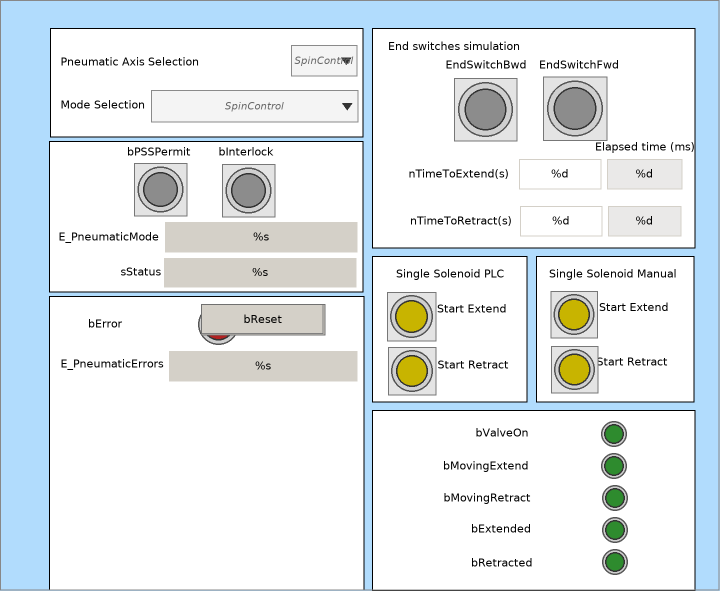
VISUALIZATION PneumaticsVisu_1  // 720x591
    Rectangle (50,28 313x109)
    Label (55,47 150x30), "Pneumatic Axis Selection"
    Rectangle (372,28 323x220)
    Label (379,30 150x33), "End switches simulation"
    Label (411,50 150x30), "EndSwitchBwd"
    SpinControl (291,45 66x31), variable: MAIN.hmiPneumaticAxisSelection
        p651134158: GVL_APP.nPNEUMATIC_AXIS_NUM
    Label (504,50 150x30), "EndSwitchFwd"
    Rectangle (49,296 315x294)
    Textfield (519,159 82x30), "%d", text variable: MAIN.afbPneumaticAxes[MAIN.hmiPneumaticAxisSelection].stPneumaticAxisStruct.stPneumaticAxisConfig.nTimeToExtend
        OnMouseClick: write MAIN.afbPneumaticAxes[MAIN.hmiPneumaticAxisSelection].stPneumaticAxisStruct.stPneumaticAxisConfig.nTimeToExtend via Default
    Label (384,159 150x30), "nTimeToExtend(s)"
    Label (386,206 150x30), "nTimeToRetract(s)"
    Label (28,90 150x30), "Mode Selection"
    Rectangle (49,141 314x151)
    Label (30,309 150x30), "bError"
    Lamp1 (126,301 185x47), variable: MAIN.afbPneumaticAxes[MAIN.hmiPneumaticAxisSelection].stPneumaticAxisStruct.stPneumaticAxisStatus.bError, style: Lamp-Lamp1-Red
    Label (37,349 150x30), "E_PneumaticErrors"
    Textfield (169,351 188x30), "%s", text variable: MAIN.afbPneumaticAxes[MAIN.hmiPneumaticAxisSelection].stPneumaticAxisStruct.ePneumaticAxisErrors, text list: 'languageSupport'
    Rectangle (372,256 155x146)
    Rectangle (536,256 158x146)
    Rectangle (372,410 323x181)
    Label (538,259 150x30), "Single Solenoid Manual"
    PushSwitchLed (549,291 50x47), variable: MAIN.afbPneumaticAxes[MAIN.hmiPneumaticAxisSelection].stPneumaticAxisStruct.stPneumaticAxisInputs.bOpenManual, behaviour: TOGGLE, style: Switch-PushSwitchLed-Yellow
    Label (592,293 84x29), "Start Extend"
    Label (557,347 150x30), "Start Retract"
    Label (375,259 150x30), "Single Solenoid PLC"
    PushSwitchLed (387,292 49x49), variable: MAIN.afbPneumaticAxes[MAIN.hmiPneumaticAxisSelection].stPneumaticAxisStruct.stPneumaticAxisControl.bExtend, behaviour: TOGGLE, style: Switch-PushSwitchLed-Yellow
    PushSwitchLed (388,347 48x48), variable: MAIN.afbPneumaticAxes[MAIN.hmiPneumaticAxisSelection].stPneumaticAxisStruct.stPneumaticAxisControl.bRetract, behaviour: TOGGLE, style: Switch-PushSwitchLed-Yellow
    Label (427,418 150x30), "bValveOn"
    Lamp1 (539,419 150x30), variable: MAIN.afbPneumaticAxes[MAIN.hmiPneumaticAxisSelection].stPneumaticAxisStruct.stPneumaticAxisOutputs.bValveOn, style: Lamp-Lamp1-Green
    Label (411,451 150x30), "bMovingExtend"
    Lamp1 (539,451 150x30), variable: MAIN.afbPneumaticAxes[MAIN.hmiPneumaticAxisSelection].stPneumaticAxisStruct.stPneumaticAxisStatus.bExtending, style: Lamp-Lamp1-Green
    Lamp1 (540,483 150x30), variable: MAIN.afbPneumaticAxes[MAIN.hmiPneumaticAxisSelection].stPneumaticAxisStruct.stPneumaticAxisStatus.bRetracting, style: Lamp-Lamp1-Green
    Lamp1 (540,515 150x30), variable: MAIN.afbPneumaticAxes[MAIN.hmiPneumaticAxisSelection].stPneumaticAxisStruct.stPneumaticAxisStatus.bExtended, style: Lamp-Lamp1-Green
    Lamp1 (540,547 150x30), variable: MAIN.afbPneumaticAxes[MAIN.hmiPneumaticAxisSelection].stPneumaticAxisStruct.stPneumaticAxisStatus.bRetracted, style: Lamp-Lamp1-Green
    Label (412,483 150x30), "bMovingRetract"
    Label (426,514 150x30), "bExtended"
    Label (397,294 150x30), "Start Extend"
    Label (398,350 150x30), "Start Retract"
    Label (427,548 150x30), "bRetracted"
    Button (201,304 124x31), "bReset"
        toggle MAIN.afbPneumaticAxes[MAIN.hmiPneumaticAxisSelection].stPneumaticAxisStruct.stPneumaticAxisControl.bReset
    PushSwitchLed (549,346 51x47), variable: MAIN.afbPneumaticAxes[MAIN.hmiPneumaticAxisSelection].stPneumaticAxisStruct.stPneumaticAxisInputs.bCloseManual, behaviour: TOGGLE, style: Switch-PushSwitchLed-Yellow
    Label (84,137 150x30), "bPSSPermit"
    Label (34,222 150x30), "E_PneumaticMode"
    Textfield (165,222 192x30), "%s", text variable: MAIN.afbPneumaticAxes[MAIN.hmiPneumaticAxisSelection].stPneumaticAxisStruct.ePneumaticAxisMode, text list: 'languageSupport'
    Textfield (164,258 192x29), "%s", text variable: MAIN.afbPneumaticAxes[MAIN.hmiPneumaticAxisSelection].stPneumaticAxisStruct.stPneumaticAxisStatus.sStatus, text list: 'languageSupport'
    Label (66,257 150x30), "sStatus"
    Textfield (520,206 82x30), "%d", text variable: MAIN.afbPneumaticAxes[MAIN.hmiPneumaticAxisSelection].stPneumaticAxisStruct.stPneumaticAxisConfig.nTimeToRetract
        OnMouseClick: write MAIN.afbPneumaticAxes[MAIN.hmiPneumaticAxisSelection].stPneumaticAxisStruct.stPneumaticAxisConfig.nTimeToRetract via Default
    Textfield (607,159 75x30), "%d", text variable: MAIN.afbPneumaticAxes[MAIN.hmiPneumaticAxisSelection].fbTimerExtend.ET
    Textfield (608,206 73x30), "%d", text variable: MAIN.afbPneumaticAxes[MAIN.hmiPneumaticAxisSelection].fbTimerRetract.ET
    SpinControl (151,90 207x32), variable: MAIN.afbPneumaticAxes[MAIN.hmiPneumaticAxisSelection].stPneumaticAxisStruct.ePneumaticAxisMode
    Label (570,132 150x30), "Elapsed time (ms)"
    PushSwitchLed (454,77 63x65), variable: MAIN.afbPneumaticAxes[MAIN.hmiPneumaticAxisSelection].stPneumaticAxisStruct.stPneumaticAxisInputs.bEndSwitchBwd, behaviour: TOGGLE, style: Switch-PushSwitchLed-Gray
    PushSwitchLed (543,76 64x65), variable: MAIN.afbPneumaticAxes[MAIN.hmiPneumaticAxisSelection].stPneumaticAxisStruct.stPneumaticAxisInputs.bEndSwitchFwd, behaviour: TOGGLE, style: Switch-PushSwitchLed-Gray
    PushSwitchLed (134,163 53x53), variable: MAIN.afbPneumaticAxes[MAIN.hmiPneumaticAxisSelection].stPneumaticAxisStruct.stPneumaticAxisInputs.bPSSPermit, behaviour: TOGGLE, style: Switch-PushSwitchLed-Gray
    PushSwitchLed (222,164 53x53), variable: MAIN.afbPneumaticAxes[MAIN.hmiPneumaticAxisSelection].stPneumaticAxisStruct.stPneumaticAxisControl.bInterlock, behaviour: TOGGLE, style: Switch-PushSwitchLed-Gray
    Label (171,137 150x30), "bInterlock"
END_VISUALIZATION

(* stored: Version 1.1.0.1, ProductVersion 3.1.4024.12
   Visu PneumaticsVisu_1: Id {ae23f543-ccab-4934-bfc1-920eae821ebc} *)
